// TwinCAT 3 PLC project F_LogToInflux
// ProgramVersion: 3.1.4022.2
// libraries:
//   log4TC, * (mbc engineering GmbH)
//   Tc2_Standard, * (Beckhoff Automation GmbH)
//   Tc2_System, * (Beckhoff Automation GmbH)
//   Tc3_Module, * (Beckhoff Automation GmbH)
// project tree:
//   / MAIN.TcPOU, PlcTask.TcTTO
// real-time tasks:
//   TASK PlcTask: cycle T#10ms, priority 20, ADS port 350

CONFIGURATION F_LogToInflux
    RESOURCE PLC ON TwinCAT3
        TASK PlcTask(INTERVAL := T#10ms, PRIORITY := 20);
        PROGRAM MAIN WITH PlcTask : MAIN;
    END_RESOURCE
END_CONFIGURATION

// ---- MAIN.TcPOU
PROGRAM MAIN
VAR
	nCount			: UINT;
	nExecTimeSum	: UDINT;
	nExecTimeMin	: UDINT := 16#FFFFFFFF;
	nExecTimeMax	: UDINT := 0;
END_VAR
VAR_TEMP
	nExecTimeAvg	: UDINT;
END_VAR

IF _TaskInfo[GETCURTASKINDEXEX()].FirstCycle THEN
	// For Remote Log4TC Server change the AMS net ID and configure a route
	PRG_TaskLog.Init('127.0.0.1.1.1');
	F_Log(E_LogLevel.eInfo, 'SPS Task gestartet.');
END_IF

nExecTimeSum := nExecTimesum + _TaskInfo[1].LastExecTime;
nExecTimeMax := MAX(nExecTimeMax, _TaskInfo[1].LastExecTime);
nExecTimeMin := MIN(nExecTimeMin, _TaskInfo[1].LastExecTime);
nCount := nCount + 1;

IF (nCount * _TaskInfo[1].CycleTime) >= (1 * 10000000) THEN
	nExecTimeAvg := nExecTimeSum / nCount;
	F_LogLA3(
		E_LogLevel.eTrace,
		'influxdb.cycletime',
		'Cycle time: {avg}/{min}/{max}',
		nExecTimeAvg,
		nExecTimeMin,
		nExecTimeMax
	);
	
	nExecTimeSum := 0;
	nExecTimeMin := 16#FFFFFFFF;
	nExecTimeMax := 0;
	nCount := 0;
END_IF

PRG_TaskLog.Call();

END_PROGRAM
